Universal Robots URScript: suspension_script_experiment.script

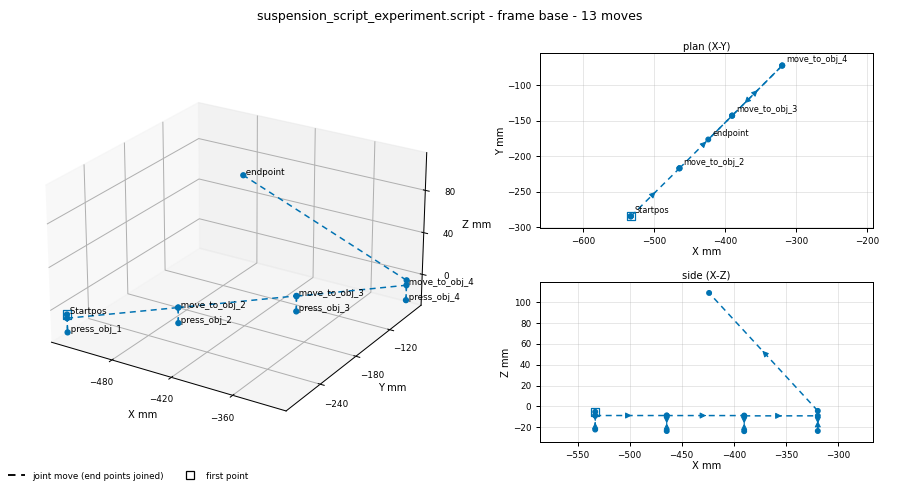
[picture p0: tool path of suspension_script_experiment.script in frame base, 13 of 13 moves have a stored position in this frame; points joined in program order, loops and branches not executed]
def suspension_script_experiment():
  step_count_d155977c_0a41_48ae_bd27_7c6c2596e01b = 0.0
  thread Step_Counter_Thread_a49c3dc3_a476_4b70_9abb_93f09a6f83ec():
    while (True):
      step_count_d155977c_0a41_48ae_bd27_7c6c2596e01b = step_count_d155977c_0a41_48ae_bd27_7c6c2596e01b + 1.0
      sync()
    end
  end
  run Step_Counter_Thread_a49c3dc3_a476_4b70_9abb_93f09a6f83ec()
  set_tool_communication(False, 115200, 0, 1, 1.5, 3.5)
  set_tool_output_mode(0)
  set_tool_digital_output_mode(0, 1)
  set_tool_digital_output_mode(1, 1)
  set_tool_voltage(0)
  set_standard_analog_input_domain(0, 1)
  set_standard_analog_input_domain(1, 1)
  set_tool_analog_input_domain(0, 1)
  set_tool_analog_input_domain(1, 1)
  set_analog_outputdomain(0, 0)
  set_analog_outputdomain(1, 0)
  set_input_actions_to_default()
  set_safety_mode_transition_hardness(1)
  set_gravity([0.0, 0.0, 9.82])
  set_tcp(p[0.0,0.0,0.184,0.0,0.0,0.0])
  set_target_payload(1.500000, [0.000000, -0.002000, 0.046000], [0.003026, 0.003026, 0.003026, 0.000000, 0.000000, 0.000000])
  global Line_1=p[0.0,0.0,0.0,0.0,0.0,0.0]
  global Line_2=p[0.0,0.0,0.0,0.0,0.0,0.0]
  global Plane_1=p[-0.361487432735338,-0.016717979378191757,0.10394933298158474,0.8032803749589464,-1.48273794275507,-1.3712545351254601]
  global Plane_2=p[-0.4390181010417212,-0.5025363244384129,0.07754186088006663,0.0242452931196319,-0.008431548293163078,-0.5708956925038724]
  global Plane_3=p[-0.25480483753173705,-0.5081372437231373,0.07201538765959875,-9.039930063647936E-5,-1.434349324572951E-4,-0.3090720642039013]
  global Point_3=p[0.0,0.0,0.0,0.0,0.0,0.0]
  global floorgripper=p[-0.2464960731348849,-0.4897452928079739,0.0709944577944641,1.7320762453741406E-4,5.47703051263464E-6,-0.32694642097279897]
  global front_collision=p[-0.4941642762715196,-0.6127463334128198,0.7662532960153384,1.5,4.484756383203096E-16,2.3363997805214006E-16]
  global table=p[-0.8492357722348507,-0.0703668253590126,-0.04045,-2.900828785048298,-1.2031999063950631,-7.106365334326772E-4]
  # begin: URCap Installation Node
  #   Source: External Control, 1.0.5, FZI Research Center for Information Technology
  #   Type: External Control
  # end: URCap Installation Node
  global Startpos_p=p[-.532996777216, -.284744003193, -.005258658650, -.041335465478, 3.127948677547, .035148430359]
  global Startpos_q=[0.2755400836467743, -1.0811593395522614, 1.7971132437335413, -2.2670165501036585, -1.5881403128253382, -1.3223417440997522]
  global press_obj_1_p=p[-.533016647477, -.284741041138, -.022262376561, -.041372693237, 3.127987940013, .035147110842]
  global press_obj_1_q=[0.275515079498291, -1.0535686773112793, 1.8085368315326136, -2.3060690365233363, -1.5881412664996546, -1.32233173051943]
  global release_obj_1_p=p[-.533004454871, -.284724041167, -.008800510653, -.041296838723, 3.127947770957, .035111853913]
  global release_obj_1_q=[0.27549031376838684, -1.075529770260193, 1.799657169972555, -2.2751947842040003, -1.5881155172931116, -1.322355095540182]
  global move_to_obj_2_p=p[-.464337053823, -.216959997013, -.008814231925, -.041387927723, 3.127949251703, .035130040595]
  global move_to_obj_2_q=[0.18425607681274414, -1.245681033735611, 2.073148552571432, -2.3802806339659632, -1.5890753904925745, -1.4138239065753382]
  global press_obj_2_p=p[-.464336433556, -.216966524036, -.023690949031, -.041293704885, 3.127967092241, .035140669214]
  global press_obj_2_q=[0.18425500392913818, -1.2156447631171723, 2.084029022847311, -2.4212104282774867, -1.589074436818258, -1.4136789480792444]
  global release_obj_2_p=p[-.464330106405, -.216952356473, -.008835163881, -.041350405827, 3.127913706779, .035137852585]
  global release_obj_2_q=[0.18424296379089355, -1.2456456881812592, 2.073160950337545, -2.38029207805776, -1.589074436818258, -1.4138129393206995]
  global move_to_obj_3_p=p[-.389969660679, -.142624736729, -.008849024720, -.041444059103, 3.127896307941, .035184358364]
  global move_to_obj_3_q=[0.0392039529979229, -1.438633458023407, 2.3400681654559534, -2.457254549066061, -1.5907309691058558, -1.5592225233661097]
  global press_obj_3_p=p[-.389986347474, -.142633985660, -.023852823447, -.041456378506, 3.127974322820, .035175940922]
  global press_obj_3_q=[0.03919276222586632, -1.3990323108485718, 2.3534629980670374, -2.5103260479369105, -1.5907066504107874, -1.5591033140765589]
  global release_obj_3_p=p[-.389938014959, -.142625330573, -.009120125990, -.041388781142, 3.127849026216, .035148719282]
  global release_obj_3_q=[0.03919126093387604, -1.4379886996797104, 2.3403692881213587, -2.4581524334349574, -1.5907066504107874, -1.559197727833883]
  global move_to_obj_4_p=p[-.319305747377, -.071938578125, -.009098739514, -.041345570106, 3.127950334567, .035097416430]
  global move_to_obj_4_q=[-0.17440492311586553, -1.653053422967428, 2.5667811075793665, -2.4746090374388636, -1.5926597754107874, -1.7732890287982386]
  global press_obj_4_p=p[-.319322901862, -.071914273425, -.023663041840, -.041252472099, 3.127989201398, .035207760819]
  global press_obj_4_q=[-0.17446500459779912, -1.6011196575560511, 2.583975378667013, -2.543784280816549, -1.592673126851217, -1.7730844656573694]
  global release_obj_4_p=p[-.319306728102, -.071929629451, -.004335743919, -.041338714269, 3.127978018768, .035193643440]
  global release_obj_4_q=[-0.1743691603290003, -1.6691600284972132, 2.560770336781637, -2.452531953851217, -1.5927332083331507, -1.7733119169818323]
  global endpoint_p=p[-.423662398290, -.176278308356, .108875172493, -.041332781470, 3.128003211959, .035136268584]
  global endpoint_q=[0.11230076104402542, -1.5612164328670879, 2.0770867506610315, -2.0702268085875453, -1.5902369658099573, -1.4865496794330042]
  while (True):
    $ 1 "Robot Program"
    $ 2 "MoveJ"
    $ 3 "Startpos" "breakAfter"
    movej(get_inverse_kin(Startpos_p, qnear=Startpos_q), a=1.3962634015954636, v=1.0471975511965976)
    $ 4 "MoveJ"
    $ 5 "press_obj_1" "breakAfter"
    movej(get_inverse_kin(press_obj_1_p, qnear=press_obj_1_q), a=1.3962634015954636, v=1.0471975511965976)
    $ 6 "MoveJ"
    $ 7 "release_obj_1" "breakAfter"
    movej(get_inverse_kin(release_obj_1_p, qnear=release_obj_1_q), a=1.3962634015954636, v=1.0471975511965976)
    $ 8 "MoveJ"
    $ 9 "move_to_obj_2" "breakAfter"
    movej(get_inverse_kin(move_to_obj_2_p, qnear=move_to_obj_2_q), a=1.3962634015954636, v=1.0471975511965976)
    $ 10 "MoveJ"
    $ 11 "press_obj_2" "breakAfter"
    movej(get_inverse_kin(press_obj_2_p, qnear=press_obj_2_q), a=1.3962634015954636, v=1.0471975511965976)
    $ 12 "MoveJ"
    $ 13 "release_obj_2" "breakAfter"
    movej(get_inverse_kin(release_obj_2_p, qnear=release_obj_2_q), a=1.3962634015954636, v=1.0471975511965976)
    $ 14 "MoveJ"
    $ 15 "move_to_obj_3" "breakAfter"
    movej(get_inverse_kin(move_to_obj_3_p, qnear=move_to_obj_3_q), a=1.3962634015954636, v=1.0471975511965976)
    $ 16 "MoveJ"
    $ 17 "press_obj_3" "breakAfter"
    movej(get_inverse_kin(press_obj_3_p, qnear=press_obj_3_q), a=1.3962634015954636, v=1.0471975511965976)
    $ 18 "MoveJ"
    $ 19 "release_obj_3" "breakAfter"
    movej(get_inverse_kin(release_obj_3_p, qnear=release_obj_3_q), a=1.3962634015954636, v=1.0471975511965976)
    $ 20 "MoveJ"
    $ 21 "move_to_obj_4" "breakAfter"
    movej(get_inverse_kin(move_to_obj_4_p, qnear=move_to_obj_4_q), a=1.3962634015954636, v=1.0471975511965976)
    $ 22 "MoveJ"
    $ 23 "press_obj_4" "breakAfter"
    movej(get_inverse_kin(press_obj_4_p, qnear=press_obj_4_q), a=1.3962634015954636, v=1.0471975511965976)
    $ 24 "MoveJ"
    $ 25 "release_obj_4" "breakAfter"
    movej(get_inverse_kin(release_obj_4_p, qnear=release_obj_4_q), a=1.3962634015954636, v=1.0471975511965976)
    $ 26 "MoveJ"
    $ 27 "endpoint" "breakAfter"
    movej(get_inverse_kin(endpoint_p, qnear=endpoint_q), a=1.3962634015954636, v=1.0471975511965976)
  end
end
